// TIA Portal V19 export
FUNCTION "STD_UPDATE_STEP_OP25" : Void   // FC3, STL
{ S7_Optimized_Access := 'TRUE' }
AUTHOR : JOM
FAMILY : STD
NAME : UPD_STEP
// stored: AutoNumber false
   VAR_INPUT
      START : Bool;
      FLAG_WORD : Int;
      OFFSET : Int;
      MAX : Int;
      MAIN_NO : Int;
   END_VAR
   VAR_IN_OUT
      OLD_STATUS : Word;
      COUNT : Int;
      MAIN : Int;
   END_VAR
   VAR_TEMP
      PUSH_REG : Int;
   END_VAR
BEGIN

NETWORK
TITLE = 
      AN    #START;
      BEC;

      L     #OLD_STATUS;
      L     #FLAG_WORD;
      ==I;
      BEC;

      L     #MAIN_NO;
      T     #MAIN;

      L     #OFFSET;
      T     #COUNT;

      L     #FLAG_WORD;
      T     "mw210_DW";
      L     "Tag_50";
      T     "Tag_51";
      L     "Tag_52";
      T     "Tag_53";

      L     "mw212_DW";
      T     #PUSH_REG;
      T     #OLD_STATUS;

LOOP: L     #PUSH_REG;
      SRW   1;
      T     #PUSH_REG;

      L     #COUNT;
      +     1;
      T     #COUNT;
      L     #OFFSET;
      -I;
      L     #MAX;
      >I;
      JC    END;

      L     #PUSH_REG;
      L     0;
      <>I;
      JC    LOOP;
      BEU;
END:  L     200;
      T     #COUNT;
      BEU;
END_FUNCTION
